// TIA Portal V17 export
// export: Created 2025-06-26T06:49:16.1420126Z, ExportSetting WithDefaults, DisplayName Totally Integrated Automation Portal, DisplayVersion V17 Update 8, DisplayName TIA Portal Openness, DisplayVersion V17 Update 8, DisplayName TIA Portal Version Control Interface, DisplayVersion V17, DisplayName STEP 7 Professional, DisplayVersion V17 Update 8, DisplayName STEP 7 Safety, DisplayVersion V17 Update 6, DisplayName WinCC Advanced, DisplayVersion V17 Update 8
FUNCTION_BLOCK "fbEvent"   // FB29, LAD
TITLE = Basic alarm
{ S7_Optimized_Access := 'TRUE' }
VERSION : 0.1
// stored: AutoNumber true, IsIECCheckEnabled false, IsRetainMemResEnabled false, MemoryReserve 0, SetENOAutomatically false, UDAEnableTagReadback false
   VAR_INPUT
      bInput : Bool;
      bAck : Bool;
      bEnable : Bool;
   END_VAR
   VAR_IN_OUT
      bActive : Bool;
      bActiveUnack : Bool;
   END_VAR
   VAR
      mActive : Bool;
   END_VAR
   VAR_TEMP   // added for the SCL form of the ladder/FBD networks
      _w1 : Bool;
   END_VAR
BEGIN

REGION Network 1: Alarm: reset if alarm is disabled or the alarm condition has cleared
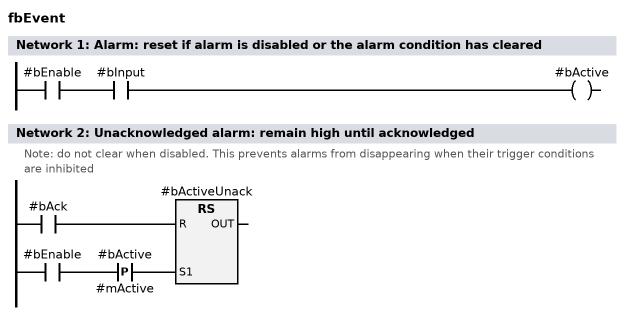
   RUNG wire#powerrail
      Contact( #bEnable )
      Contact( #bInput )
      Coil( #bActive )
   END_RUNG
   // the same network as SCL:
   #bActive := #bEnable AND #bInput;
END_REGION

REGION Network 2: Unacknowledged alarm: remain high until acknowledged
   // Note: do not clear when disabled. This prevents alarms from disappearing when their trigger conditions are inhibited
   RUNG wire#powerrail
      Contact( #bAck )
      S_RS(operand := #bActiveUnack, s1 := wire#w1)
   END_RUNG
   RUNG wire#powerrail
      Contact( #bEnable )
      P_Contact(operand := #bActive, bit := #mActive)
   END_RUNG wire#w1
   // the same network as SCL:
   #_w1 := #bEnable AND #bActive AND NOT #mActive;   // rising edge of #bActive
   #mActive := #bActive;
   IF #bAck THEN
       #bActiveUnack := FALSE;   // RS flip-flop
   END_IF;
   IF #_w1 THEN #bActiveUnack := TRUE; END_IF;
END_REGION
END_FUNCTION_BLOCK
